// TIA Portal V18 export
FUNCTION_BLOCK "TON_seconds"   // FB8, FBD
{ S7_Optimized_Access := 'TRUE' }
VERSION : 0.1
// stored: AutoNumber true, IsIECCheckEnabled false, IsRetainMemResEnabled false, MemoryReserve 100, SetENOAutomatically false, UDAEnableTagReadback false
   VAR_INPUT
      IN : Bool;
      PT_s : DInt;
   END_VAR
   VAR_OUTPUT
      Q : Bool;
   END_VAR
   VAR
      ton { S7_SetPoint := 'True'} : TON_TIME;
   END_VAR
   VAR_TEMP
      PT : Time;
   END_VAR
BEGIN

REGION Network 1
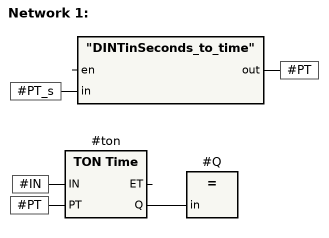
   "DINTinSeconds_to_time"(in := #PT_s, out => #PT);
   #ton(IN := #IN, PT := #PT);   // TON
   #Q := #ton.Q;
END_REGION
END_FUNCTION_BLOCK
